Universal Robots URScript: MAINTE_6001.script

def MAINTE_6001():
  global _hidden_verificationVariable=0
  step_count_9f81c29c_5f5d_49bc_9616_a2740b58e324 = 0.0
  thread Step_Counter_Thread_9d8d3198_8e35_44c5_8692_22ed9e220d66():
    while (True):
      step_count_9f81c29c_5f5d_49bc_9616_a2740b58e324 = step_count_9f81c29c_5f5d_49bc_9616_a2740b58e324 + 1.0
      sync()
    end
  end
  run Step_Counter_Thread_9d8d3198_8e35_44c5_8692_22ed9e220d66()
  set_target_payload(0.100000, [0.135000, 0.000000, 0.225000], [10.000000, 10.000000, 10.000000, 0.000000, 0.000000, 0.000000])
  set_tool_communication(False, 115200, 0, 1, 1.5, 3.5)
  set_tool_output_mode(0)
  set_tool_digital_output_mode(0, 1)
  set_tool_digital_output_mode(1, 1)
  set_tool_voltage(0)
  set_standard_analog_input_domain(0, 1)
  set_standard_analog_input_domain(1, 1)
  set_tool_analog_input_domain(0, 1)
  set_tool_analog_input_domain(1, 1)
  set_analog_outputdomain(0, 0)
  set_analog_outputdomain(1, 0)
  set_input_actions_to_default()
  set_runstate_gp_boolean_output_to_value(0, 3)
  set_tcp(p[0.0,0.08,0.42,0.0,0.0,0.0])
  set_gravity([0.0, 0.0, 9.82])
  set_safety_mode_transition_hardness(1)
  global DistPillar=339
  global CandCnt=8
  global lr=1
  global ReCaptZ=0
  global port=3000
  global socket_timeout=120
  global host="192.168.1.2"
  global is_popup=False
  global pBucket=[p[0.8599, 0.4614, 0.34265, 0, 0, -1.56701], p[-0.80901, -0.49062, 0.31822, -0, 0, 1.56854], p[0, 0, 0, 0, 0, 0]]
  global CaptStepZ=0.085
  global CaptIndex=[0, 0, 0]
  global pBucketM=p[-0.76064, -0.49997, 0.35503, 0, 0, 1.57135]
  global socket_name="vt"
  global rovi_err=0
  global SubPrgResult=100
  global CurrPos=p[-0.00403, -0.41063, 0.52839, -0.02298, -3.14138, -0.00117]
  global CurrPos_p=p[-0.00291, -0.33032, 0.10845, -0.02298, -3.14138, -0.00117]
  global ForceStartZ=0.39693
  global CutOffZ=0.08
  global HomeDistTh=0.05
  global RBDistTh=0.05
  global RBRadiusTh=0.3
  global RBXTh=[-0.5, 0.5]
  global RBYTh=[-0.8, 1]
  global RBZTh=[-0.1, 0.1]
  global Sub3100_ZMax=0.74
  global ForceStartX=-0.90368
  global Sub3100_aRot=0.2
  global Sub3100_d=0.3
  global Sub3100_Option=1
  global Sub3100_a=0.2
  global Sub3100_XdV=0.1
  global Sub3100_XdRot=8
  global ZoneDistTh=0.05
  global ZoneRadiusTh=0.3
  global ZoneXTh=[-0.5, 0.5]
  global ZoneYTh=[-0.8, 1]
  global ZoneZTh=[-0.1, 0.1]
  global BucketWidth=0.95
  global ZoneBucketGap=0
  global ZoneHomeX=0.2
  global UnloadZ=0.05
  global CaptPos=p[0.47573, -0.4259, 0.04497, 3.14138, 0.03448, 0.00005]
  global BucketUpperPos=p[0.47573, -0.4259, 0.04497, 3.14138, 0.03448, 0.00005]
  global Sub3100_GPII18=1
  global Zone6ThX=0.1
  global Zone6ThY=0.05
  global pCV=p[-0.00228, -0.00072, 0.00263, 0.00249, 0.0013, 0.00219]
  global CaptRowNo=1
  global CrankDepthFull=0.025
  global CrankDepth=0.07906
  global DistPillarTh=200
  global Y1=[0,0,0,0]
  global Y2=p[0.0,0.0,0.0,0.0,0.0,0.0]
  global Bucket=p[0.32604,0.49174,0.0,-1.882900624652718E-5,2.8304179127934987E-5,-1.593185305749222]
  global BucketM=p[0.32604,0.49174,0.0,2.2353980716304163E-16,-3.5868426080024975E-16,-1.5931853071795856]
  global CV=p[0.0,0.0,0.0,0.0,0.0,0.0]
  global CaptPoint_C=p[-0.335,-0.024,0.4,-2.196299060524223,-2.2462891909035143,-5.664484063487096E-5]
  global CaptPoint_C2=p[0.32796661698047924,-0.010768520544682924,0.01931625281283378,2.2288103429550152,-2.213636886217198,8.598462540813273E-5]
  global CaptPoint_L=p[-0.335,-0.246,0.4,-2.1962012732824228,-2.246352675070566,-1.646578372162058E-4]
  global CaptPoint_L2=p[0.327894307417917,-0.010799940826224014,0.01928712668893995,2.087717047309385,-2.0736781215133306,0.27365839887453103]
  global CaptPoint_R=p[-0.335,0.246,0.4,-2.1963444166345645,-2.2462256265309297,2.4676186941162578E-5]
  global CaptPoint_R2=p[0.327926308680866,-0.010795166414457658,0.019300245403843563,-2.1186306375223185,2.1040550557443427,0.22023197678473694]
  global Capt_1BK_L=p[-0.395,-0.47,0.35,-2.1961210242572884,-2.2463362846055,-2.908274762447041E-4]
  global Capt_1BK_R=p[-0.395,0.51,0.35,2.196067754706757,2.246288285862388,2.8411291050601595E-5]
  global Capt_1BK_pos1=p[-0.4218793038724447,-0.003154429464978058,0.2915499891144615,-2.1963422029204875,-2.2438663520270015,-0.02197160668673838]
  global Capt_1BK_pos2=p[-0.42187829024618434,-0.0031710253373066375,0.29156503858953065,-2.196324918349679,-2.2439040699490773,-0.021928444416953782]
  global Capt_2BK_L=p[0.42186661528427194,0.4254738068040517,0.35042275762909847,2.239156309475874,-2.1837044610999294,0.002643817066643282]
  global Capt_2BK_R=p[0.4218208572756906,-0.5427676723257963,0.350372239919558,2.2392697861179327,-2.183553596194912,0.002410470905346486]
  global Capt_2BK_pos1=p[0.42193501458435656,0.004742683868356356,0.35045865974037793,2.2391012408536453,-2.1839704655717003,0.002677867056024068]
  global Capt_2BK_pos2=p[0.421903984494575,0.004707988774967922,0.35045218900915065,2.239114367170047,-2.183895515396197,0.002684056681074047]
  global Capt_CV_M=p[-0.04794223960540197,-0.559868557160475,0.1086937653706071,-0.022464429848058916,-3.141454018347238,4.0166993855964835E-4]
  global Capt_GD_M=p[-0.004053197679954899,-0.25261725691632436,-0.01970497430780127,0.0332779454553888,-3.140179196376707,-0.0034093680964018282]
  global HomePointL=p[-0.36789,-0.5117344641471838,0.78,-0.6278857271586024,3.0680899128661667,-8.649957362498864E-4]
  global Master_pos=p[-0.002900061250386237,-0.3308544176418705,0.08247088152898924,-0.022398151655969412,-3.1414279476897704,4.608357258864606E-4]
  global PickPos=p[0.10830682331105715,-1.3709505888096256,-0.18404188875951455,-0.00622194000158997,2.880236948927292,-0.00383636509397631]
  global Solve=p[-0.00368,-0.0021000000000000003,0.25739999999999996,0.0,0.0,0.0]
  global TCP3100TL=p[0.0,0.06,0.535,1.8939999999999997,0.0,0.0]
  global TEST=p[0.1,0.0,0.2,0.0,0.0,0.0]
  global UF=p[0.0,0.0,0.0,0.0,0.0,0.0]
  global g1CV_posL1=p[0.05028133628211688,-0.4526481033729615,0.1221845548632916,-2.213335080948508,-2.1937561336067057,-0.3280056759040735]
  global g1CV_posR1=p[0.03743870476062511,-0.53119407812668,0.11301901343688614,2.073418671558482,2.153257467049566,0.11656306439039889]
  global g1GD_pos1=p[0.14857012745627257,-0.6379982996093139,0.2691918735517042,2.214277610229479,2.228493098198348,-1.6896832945346036E-4]
  global g1GD_pos2=p[0.028634297882679793,-0.4702313285867709,0.450031657325677,2.214319081558633,2.2285182736309666,-1.5473710223511705E-5]
  global g1GD_pos3=p[-0.1945307709581842,-0.42906455111749103,0.45,-2.685709191057467,-1.6297557787554324,7.112239955701245E-5]
  global g1GD_pos4=p[-0.25628841794770224,-0.020630481098425146,0.45,2.148716725221303,2.2918109407224354,-1.3854918368741778E-5]
  global g1GD_pos5=p[-0.714365317693782,-0.022971007293656684,0.45,-2.1476725881724037,-2.292771958266831,6.311233907547867E-5]
  global g1GD_posL1=p[-0.08276848269606216,-0.3996147100031649,0.1488453551331823,2.286527078917204,1.8420745504477611,0.33698451773695576]
  global g1GD_posL2=p[-0.3253977027403738,-0.3024804624281039,0.16332814085945146,2.72312820760317,0.9631021078169197,0.32447452035226126]
  global g1GD_posL3=p[-0.6791033397183219,0.06787475590683856,0.16337212788108813,2.1383125299263996,2.086116032377724,0.4536080263755059]
  global g1GD_posR1=p[-0.09893370538053747,-0.4999608954567234,0.14329885217724153,2.43311852414254,1.4238397520832589,0.08559216753941556]
  global g1GD_posR2=p[-0.3729565201882258,-0.3752983669473301,0.143299052800563,2.6951655216297596,0.8130506811102118,-0.02387549506099888]
  global g1GD_posR3=p[-0.7385929502572233,-0.029472684480355026,0.1499650660949685,2.0484522752014467,1.9493695704119496,0.18368227556562683]
  global g2CV_posL1=p[0.3409386496330911,-0.4656338066361442,0.1250074988128972,2.209372209162659,2.1945371304665926,0.3160714960040194]
  global g2CV_posR1=p[0.3400736278759575,-0.531334269888987,0.1183415684753657,2.07314649492589,2.1532617466521136,0.11638666128062146]
  global g2GD_pos1=p[0.2541383831722086,-0.6774928758666339,0.18519960582577166,-2.0375719953016755,-2.3889847960447277,-0.0020926217702447064]
  global g2GD_pos2=p[0.2548303032832998,-0.4395886120507379,0.2986557393825452,-1.8691601740155521,-2.5210138137905886,-0.00387894312889377]
  global g2GD_pos3=p[0.3379879014596998,-0.06467509721500111,0.3,-0.13681955358471554,3.138134920213652,0.0052602971824959885]
  global g2GD_pos4=p[0.31412137931928874,0.14047894136547145,0.3,1.0726627132331576,-2.952135651121033,-0.005044331815994264]
  global g2GD_pos5=p[0.596826867485263,0.012800854207951809,0.3,-2.250960447020382,2.191482163995288,-8.62049956035814E-5]
  global gCV_11_M=p[0.27458092838097625,-0.9634709900409619,-0.027246106999398,2.1579958677359365,2.061920489504824,0.29122365164018676]
  global gCV_12_M=p[0.32374082043819774,-0.9643905557999398,-0.025487605485889797,2.171002695191275,2.0268053402328294,0.3318967209792993]
  global gCV_13_M=p[0.3677028242565019,-0.8912043588518235,0.06406475497489328,2.0725171273330782,1.9964853271438565,0.36457536397978224]
  global gCV_1_M=p[0.2542346432653502,-0.9630040614242789,-0.02334867377482014,2.2207135850363673,2.222089414386077,-1.1830719805507357E-4]
  global gCV_2_M=p[0.2533471161659082,-0.9538280156244117,0.053347089211651155,2.2211302871500327,2.221672468159851,6.057343292863739E-5]
  global gCV_3_M=p[0.29099390607376485,-0.6570558385379063,0.0722153583041818,1.9884242634571576,2.2321538498123994,0.15249643504377583]
  global gCV_pos5=p[0.3400172856834047,-0.9722754606605235,-0.18287928563575456,2.073394561413637,2.1531827558666565,0.11639000988241816]
  global gGD_1_LM=p[0.023694495567209206,-0.7289549597812236,-0.114436637727933,-0.010169347158913183,2.8707671818561686,0.2884627079222755]
  global gGD_1_M=p[0.023465033498111344,-0.7266069947313496,-0.114063572547692,-0.02957171388996286,-3.1242906749658705,-0.31017837385641756]
  global gGD_1_RM=p[0.02362723078317132,-0.7265300624800513,-0.11281451079208593,-0.06253229749015159,-2.8808212567082383,-0.28238046714011716]
  global gGD_2_LM=p[0.024174132054917155,-0.6705540375362067,-0.11458821415948689,-0.01017914088038848,2.87086541323498,0.2882827167190487]
  global gGD_2_M=p[0.023891548276160204,-0.6721896307283143,-0.11405798252635202,-0.029537226830795685,-3.1242353369640576,-0.3100661332499525]
  global gGD_2_RM=p[0.02429249604336059,-0.6691638128218599,-0.11302949794491796,-0.06253008389277033,-2.8809170794832206,-0.2823080231602885]
  global gGD_3_LM=p[0.02414949255188298,-0.6344183862527816,-0.0037208795646377912,-0.010168403617012718,2.8708622039997236,0.2881723112066594]
  global gGD_3_M=p[0.023938978441106873,-0.6361306661281794,-0.005216445129412717,-0.029429851638448117,-3.124169609374898,-0.3100490421418616]
  global gGD_3_RM=p[0.02427953911879352,-0.6347229115915235,-0.00845845992375066,-0.062415244957792,-2.8809080008278363,-0.2823877130468298]
  global gGD_4_LM=p[-0.12534109989305553,-0.6345452257364079,-0.003660409912739915,-0.010209507081901941,2.87092276677584,0.2878514545752189]
  global gGD_4_RM=p[0.1741356102640685,-0.6348673415405857,-0.008407071546374267,-0.06250935255312234,-2.8810578033032743,-0.28204363282303685]
  global gHome_Position=p[-0.002884216431119573,-0.33081338952181766,0.10869836126442783,-0.022308300881783188,-3.141473239616493,3.9861399141130865E-4]
  global gTAIHI_pos1=p[0.034435296708333146,-0.2890869270984411,0.28697762766096685,-0.9517096680276043,2.9907327255336362,-0.006242657270483182]
  global gTAIHI_pos2=p[0.46041690381401934,0.09562026346103787,0.3409455343940188,-2.575428180750575,1.7504967205574518,-0.009370784990557466]
  global gTAIHI_pos3=p[0.4777514786587304,0.10855417509450788,0.25667938190447326,-3.115092130529677,-0.059113053813058626,0.017060902648732133]
  global gTAIHI_pos4=p[0.47773948064032057,0.10853581553326999,-0.15133852019421468,-3.1151611852917296,-0.05914313994407087,0.017149581050184888]
  global gTAIHI_pos5=p[0.30588450070104545,0.17870028478253597,-0.38750721344025674,-3.115302721311487,-0.05927431563397507,0.01725874757592571]
  rtde_set_watchdog("speed_slider_mask", 10.0, "ignore")
  # begin: URCap Installation Node
  #   Source: Ethernet/IP I/O Monitor URCap, 1.0.0,
  #   Type: Ethernet/IP I/O Monitor
  conn = rpc_factory("xmlrpc", "http://127.0.0.1:" + to_str(61101) + "/RPC2")

  def show_monitor():
    return conn.eip_monitor.show()
  end
  # end: URCap Installation Node
  global CaptPos0_p=p[.062940695952, -.648805201720, .499601675630, -.057956765798, 3.122671515713, .012933073207]
  global CaptPos0_q=[-1.2119177023517054, -1.5154119108668347, -1.9421818256378174, -1.2562483710101624, 1.5889158248901367, 0.3233448565006256]
  def SUB_001():
    $ 10 "SUB_001" "noBreak"
    $ 11 "荷重の設定: k10"
    set_target_payload(0.100000, [0.135000, 0.000000, 0.225000], [10.000000, 10.000000, 10.000000, 0.000000, 0.000000, 0.000000])
    $ 12 "MoveJ"
    $ 13 "gHome_Position" "breakAfter"
    set_tcp(p[0.0,0.08,0.42,0.0,0.0,0.0])
    movej(gHome_Position, a=0.5235987755982988, v=1.2217304763960306)
  end
  def SUB_6001():
    $ 14 "SUB_6001" "noBreak"
    $ 15 "荷重の設定: k10"
    set_target_payload(0.100000, [0.135000, 0.000000, 0.225000], [10.000000, 10.000000, 10.000000, 0.000000, 0.000000, 0.000000])
    $ 16 "If文 ( not ROVI_RESET())"
    if ((  not  ROVI_RESET())):
      $ 17 "SubPrgResult:=rovi_err"
      global SubPrgResult=rovi_err
      $ 18 "待機: 999999.0"
      sleep(999999.0)
    end
    $ 19 "MoveJ"
    $ 20 "CaptPos0" "breakAfter"
    set_tcp(p[0.0,0.0,0.0,0.0,0.0,0.0])
    movej(get_inverse_kin(CaptPos0_p, qnear=CaptPos0_q), a=0.20943951023931953, v=0.10471975511965977)
    $ 21 "CaptPos:=CaptPos0_p"
    global CaptPos=CaptPos0_p
    $ 22 "ループ (CaptPos[0]≠10000.0)"
    while ((CaptPos[0] != 10000.0)):
      $ 23 "MoveJ"
      $ 24 "CaptPos" "breakAfter"
      set_tcp(p[0.0,0.0,0.0,0.0,0.0,0.0])
      movej(CaptPos, a=0.20943951023931953, v=0.10471975511965977)
      $ 25 "待機: 2.0"
      sleep(2.0)
      $ 26 "If文 ( not ROVI_CAPTURE())"
      if ((  not  ROVI_CAPTURE())):
        $ 27 "SubPrgResult:=rovi_err"
        global SubPrgResult=rovi_err
        $ 28 "待機: 999999.0"
        sleep(999999.0)
      end
      $ 29 "CaptPos:=ROVI_SOLVE(is_popup=False)"
      global CaptPos=ROVI_SOLVE(is_popup=False)
    end
    $ 30 "MoveJ"
    $ 31 "CaptPos0" "breakAfter"
    set_tcp(p[0.0,0.0,0.0,0.0,0.0,0.0])
    movej(get_inverse_kin(CaptPos0_p, qnear=CaptPos0_q), a=0.20943951023931953, v=0.10471975511965977)
  end
  $ 2 "開始前シーケンス"
  $ 3 "スクリプト: ROVI_RESET.script"
  def ROVI_RESET():
    if (not socket_open(host,port,socket_name)):
      rovi_err=902
      return False
    end
    socket_send_line("X0()",socket_name)
    ret=socket_read_line(socket_name,socket_timeout)
    if (ret == "OK"):
      rovi_err=0
    elif (ret == "NG"):
      rovi_err=to_num(socket_read_line(socket_name,socket_timeout))
    else:
      ret="NG"
      rovi_err=903
    end
    socket_close(socket_name)
    if (rovi_err != 0):
      if (is_popup):
        popup(str_cat(ret,rovi_err),title="X0",warning=True,blocking=True)
      end
      return False
    else:
      return True
    end
  end
  $ 4 "スクリプト: ROVI_CAPTURE.script"
  def ROVI_CAPTURE():
  #  p=get_actual_tool_flange_pose()
    p=Bucket
    if (not socket_open(host,port,socket_name)):
      rovi_err=902
      return False
    end
    socket_send_string("X1(",socket_name)
    socket_send_string(p[0],socket_name)
    socket_send_string(",",socket_name)
    socket_send_string(p[1],socket_name)
    socket_send_string(",",socket_name)
    socket_send_string(p[2],socket_name)
    socket_send_string(",",socket_name)
    socket_send_string(p[3],socket_name)
    socket_send_string(",",socket_name)
    socket_send_string(p[4],socket_name)
    socket_send_string(",",socket_name)
    socket_send_string(p[5],socket_name)
    socket_send_line(")",socket_name)
    ret=socket_read_line(socket_name,socket_timeout)
    if (ret == "OK"):
      rovi_err=0
      f=socket_read_ascii_float(4,socket_name,socket_timeout)
      while (f[0]!=4):
        sleep(0.3)
        f=socket_read_ascii_float(4,socket_name,socket_timeout)
      end
      i=0
      while (i<4):
        Y1[i]=f[i+1]
        i=i+1
      end
    elif (ret == "NG"):
      rovi_err=to_num(socket_read_line(socket_name,socket_timeout))
    else:
      ret="NG"
      rovi_err=903
    end
    socket_close(socket_name)
    if (rovi_err != 0):
      if (is_popup):
        popup(str_cat(ret,rovi_err),title="X1",warning=True,blocking=True)
      end
      return False
    else:
      return True
    end
  end
  $ 5 "スクリプト: ROVI_SOLVE.script"
  def ROVI_SOLVE(is_popup=is_popup):
    buf=p[10000.0,0.0,0.0,0.0,0.0,0.0]
    if (not socket_open(host,port,socket_name)):
      rovi_err=902
      return False
    end
    socket_send_line("X2()",socket_name)
    ret=socket_read_line(socket_name,socket_timeout)
    if (ret == "OK"):
      rovi_err=0
      f=socket_read_ascii_float(6,socket_name,socket_timeout)
      while (f[0]!=6):
        sleep(0.3)
        f=socket_read_ascii_float(6,socket_name,socket_timeout)
      end
      counter=0
      while (counter<6):
        buf[counter]=f[counter+1]
        counter=counter+1
      end
    elif (ret == "NG"):
      rovi_err=to_num(socket_read_line(socket_name,socket_timeout))
    else:
      ret="NG"
      rovi_err=903
    end
    sleep(1.0)
    socket_close(socket_name)
    if (rovi_err != 0):
      if (is_popup):
        popup(str_cat(ret,rovi_err),title="X2",warning=True,blocking=True)
      end
    end
    return buf
  end
  $ 6 "ロボットプログラム"
  $ 7 "呼び出し SUB_001"
  SUB_001()
  $ 8 "呼び出し SUB_6001"
  SUB_6001()
  $ 9 "呼び出し SUB_001"
  SUB_001()
end
